(* Schneider Machine Expert - Basic project New project, file version 2.9.0.0 *)
(* ProjectInformations: Name=New project *)

HARDWARE
  Cpu 0: TM221CE24R
  EthernetConfiguration: NetworkName=M221, IpAllocationMode=FixedAddress, IpAddress=0.0.0.0, SubnetMask=0.0.0.0
  SerialLineConfiguration: Baud=Baud19200, Parity=ParityEven, DataBits=DataBits8, StopBits=StopBits1, PhysicalMedium=PhysicalMediumRs485, SlaveId=1, Addressing=SlaveAddressing
  MastTask: UsePeriodScanMode=false, PeriodScan=100
  FastTask: Period=255
  CpuBehavior: StartingMode=StartAsPreviousState, AutoSaveRamOnEeprom=true, WatchdogPeriod=250

SYMBOLS  (address, symbol, comment, settings)
  %I0.0     SWITCH_1
  %I0.1     SWITCH_2
  %I0.2     SWITCH_3
  %I0.3     SWITCH_4
  %I0.4     SWITCH_5
  %I0.5     SWITCH_6
  %I0.6     SWITCH_7
  %Q0.0     OUTPUT

POU New POU
  (* SectionNumber=1 *)

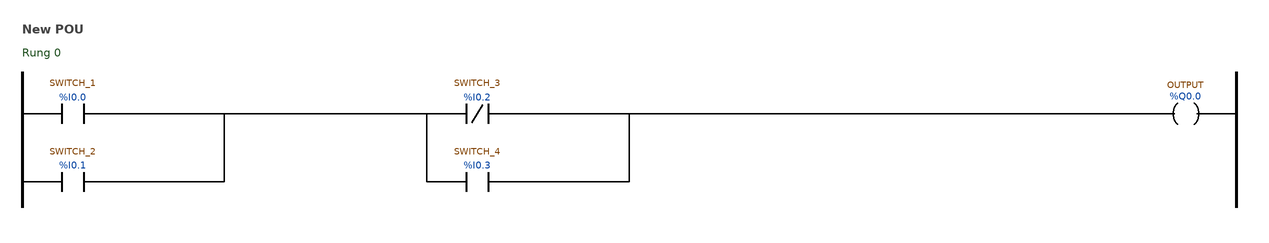

// Rung 0
  LD %I0.0                (* SWITCH_1 *)
  OR %I0.1                (* SWITCH_2 *)
  AND(N %I0.2             (* SWITCH_3 *)
  OR %I0.3                (* SWITCH_4 *)
  )
  ST %Q0.0                (* OUTPUT *)
  // as ST:
  //   OUTPUT := (SWITCH_1 OR SWITCH_2) AND (NOT SWITCH_3 OR SWITCH_4);
